Fanuc KAREL source: kb00133.KL

-- PROVISIONAL review KL for V940-1; original PC SHA256 872a72e2c90ba322adc4fafbe8038977b45f737150fe25e59b183a9c94dfc81d
-- Incomplete behavior may be omitted. Consult companion uncertainty JSON. Do not deploy.
PROGRAM KB00133
%NOLOCKGROUP
BEGIN
  -- V9_ZERO_TABLE_METADATA_HINT layout=0002_ascii; no indexed target words; source/name/runtime held
  -- UNRESOLVED_PC offsets 5-12; opcodes 9D,23
  -- UNRESOLVED_PC offsets 17-24; opcodes 9D,23
  -- UNRESOLVED_PC offsets 29-36; opcodes 9D,23
  -- UNRESOLVED_PC offsets 41-48; opcodes 9D,23
  -- UNRESOLVED_PC offsets 53-60; opcodes 9D,23
  -- UNRESOLVED_PC offsets 65-99; opcodes 27,22,22,22,22,22,31
  -- UNRESOLVED_PC offsets 104-108; opcodes 7F
END KB00133
